(* PLC project Unnamed, Unknown Unnamed 1 *)
(* stored: creationDateTime 2023-06-19T14:42:49, modificationDateTime 2023-08-09T10:28:01 *)

PROGRAM pick_and_place
  VAR
    TP0 : TP;
    CTU0 : CTU;
  END_VAR
  VAR_EXTERNAL
    ITEM_AT_ENTRY : BOOL;
    ITEM_AT_EXIT : BOOL;
    MOVING_X : BOOL;
    MOVING_Z : BOOL;
    ITEM_DETECTED : BOOL;
    START : BOOL;
    RESET : BOOL;
    STOP : BOOL;
    EMERGENCY_STOP : BOOL;
    AUTO : BOOL;
    FACTORY_IO_RUN : BOOL;
    ENTRY_CONVEYOR : BOOL;
    EXIT_CONVEYOR : BOOL;
    MOVE_X : BOOL;
    MOVE_Z : BOOL;
    GRAB : BOOL;
    START_LIGHT : BOOL;
    RESET_LIGHT : BOOL;
    STOP_LIGHT : BOOL;
    start_scada : BOOL;
    reset_scada : BOOL;
    stop_scada : BOOL;
    COUNTER : INT;
  END_VAR
  VAR
    T1_DONE : BOOL;
    TIME_DELAY : TIME := t#3s;
  END_VAR
  VAR_EXTERNAL
    STEP_0 : BOOL;
    STEP_1 : BOOL;
    STEP_2 : BOOL;
    STEP_3 : BOOL;
    STEP_4 : BOOL;
    STEP_5 : BOOL;
    STEP_6 : BOOL;
    STEP_7 : BOOL;
    STEP_LOCATION : INT;
  END_VAR
  VAR  (* added by the conversion: wires and edge detectors of the diagram *)
    R_TRIG1 : R_TRIG;
  END_VAR

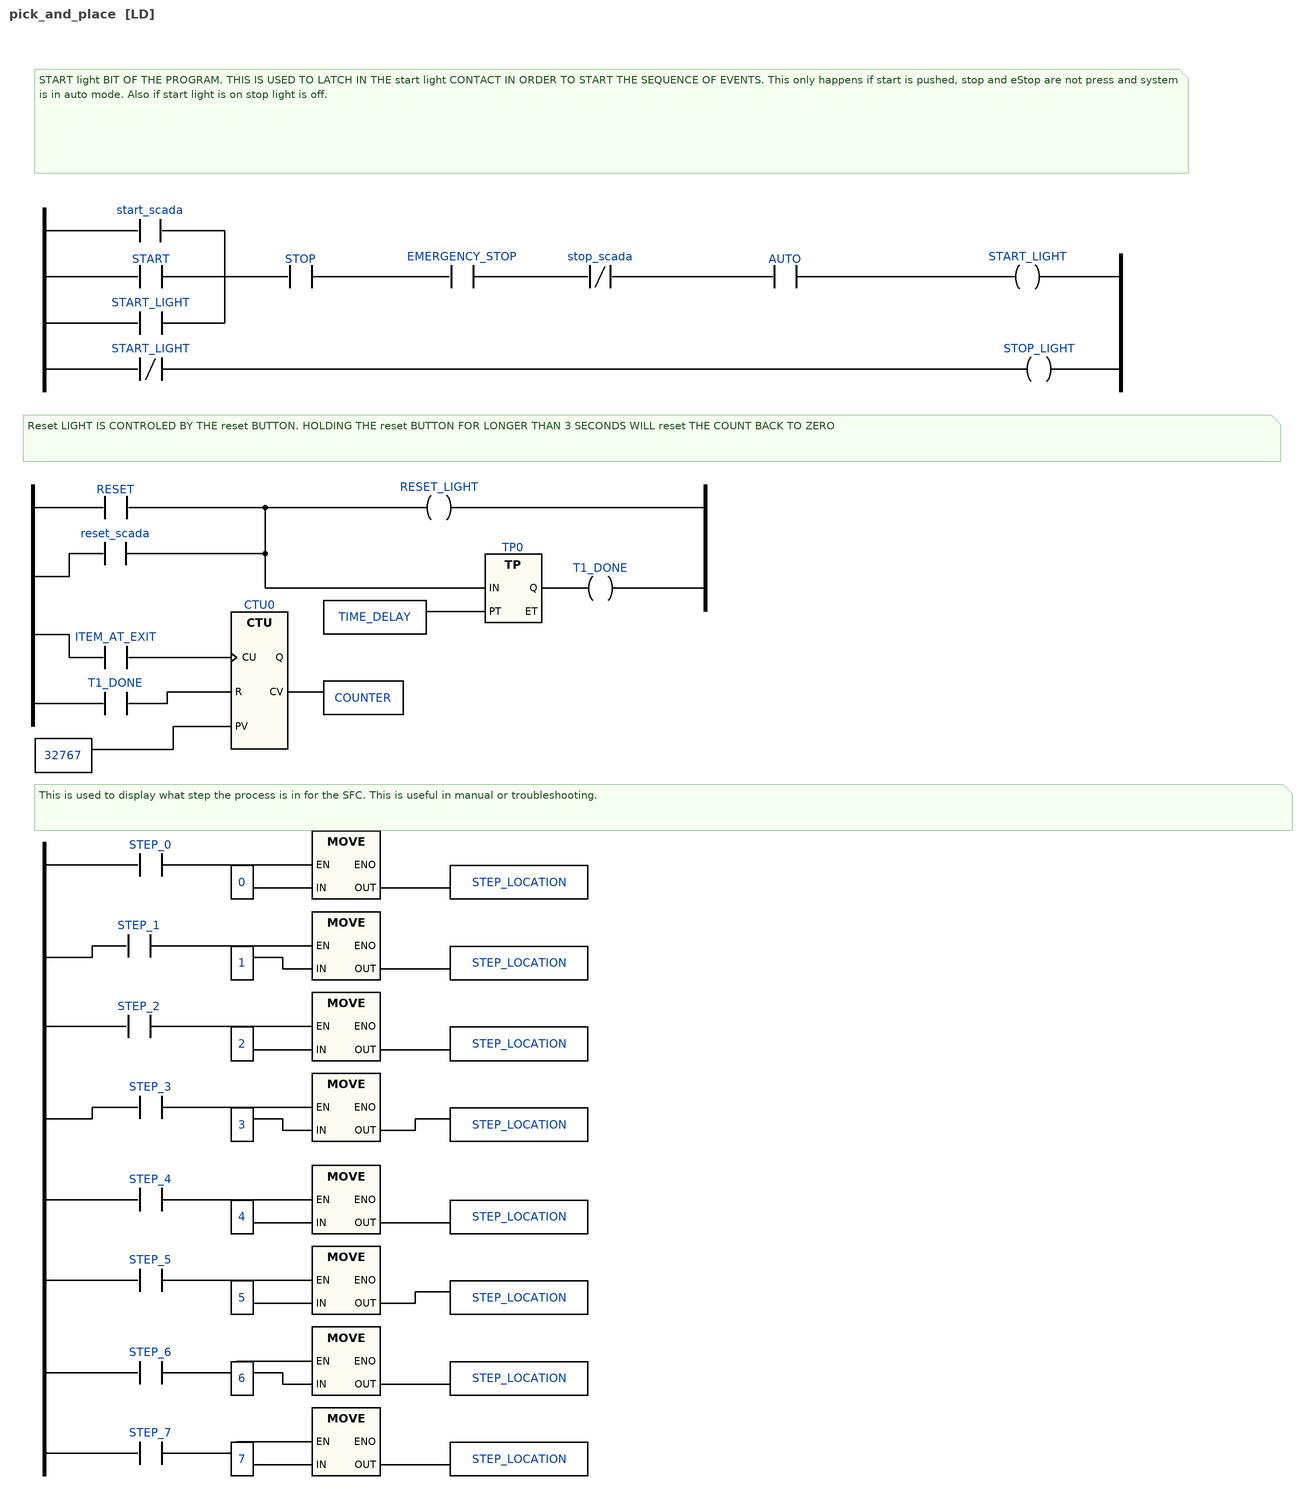
(* LD diagram, written out as Structured Text *)
(* START light BIT OF THE PROGRAM. THIS IS USED TO LATCH IN THE start light CONTACT IN ORDER TO START THE SEQUENCE OF EVENTS. This only happens if start is pushed, stop and eStop are not press and system is in auto mode. Also if start light is on stop light is off. *)
START_LIGHT := (START OR START_LIGHT OR start_scada) AND STOP AND EMERGENCY_STOP AND NOT stop_scada AND AUTO;
STOP_LIGHT := NOT START_LIGHT;
(* Reset LIGHT IS CONTROLED BY THE reset BUTTON. HOLDING THE reset BUTTON FOR LONGER THAN 3 SECONDS WILL reset THE COUNT BACK TO ZERO *)
RESET_LIGHT := RESET OR reset_scada;
TP0(IN := RESET OR reset_scada, PT := TIME_DELAY);
T1_DONE := TP0.Q;
R_TRIG1(CLK := ITEM_AT_EXIT);
CTU0(CU := R_TRIG1.Q, R := T1_DONE, PV := 32767);
COUNTER := CTU0.CV;
(* This is used to display what step the process is in for the SFC. This is useful in manual or troubleshooting. *)
IF STEP_0 THEN STEP_LOCATION := 0; END_IF;
IF STEP_1 THEN STEP_LOCATION := 1; END_IF;
IF STEP_2 THEN STEP_LOCATION := 2; END_IF;
IF STEP_3 THEN STEP_LOCATION := 3; END_IF;
IF STEP_4 THEN STEP_LOCATION := 4; END_IF;
IF STEP_5 THEN STEP_LOCATION := 5; END_IF;
IF STEP_6 THEN STEP_LOCATION := 6; END_IF;
IF STEP_7 THEN STEP_LOCATION := 7; END_IF;
END_PROGRAM

PROGRAM pick_and_place_sfc
  VAR_EXTERNAL
    ITEM_AT_ENTRY : BOOL;
    ITEM_AT_EXIT : BOOL;
    MOVING_X : BOOL;
    MOVING_Z : BOOL;
    ITEM_DETECTED : BOOL;
    START : BOOL;
    RESET : BOOL;
    STOP : BOOL;
    EMERGENCY_STOP : BOOL;
    AUTO : BOOL;
    FACTORY_IO_RUN : BOOL;
    ENTRY_CONVEYOR : BOOL;
    EXIT_CONVEYOR : BOOL;
    MOVE_X : BOOL;
    MOVE_Z : BOOL;
    GRAB : BOOL;
    START_LIGHT : BOOL;
    RESET_LIGHT : BOOL;
    STOP_LIGHT : BOOL;
    STEP_0 : BOOL;
    STEP_1 : BOOL;
    STEP_2 : BOOL;
    STEP_3 : BOOL;
    STEP_4 : BOOL;
    STEP_5 : BOOL;
    STEP_6 : BOOL;
    STEP_7 : BOOL;
    COUNTER : INT;
  END_VAR
  VAR
    R_TRIG0 : R_TRIG;
    F_TRIG0 : F_TRIG;
    F_TRIG1 : F_TRIG;
    F_TRIG2 : F_TRIG;
    F_TRIG3 : F_TRIG;
    F_TRIG4 : F_TRIG;
    F_TRIG5 : F_TRIG;
  END_VAR
  VAR  (* added by the conversion: wires and edge detectors of the diagram *)
    _SEL57_OUT : BOOL;
    _SEL61_OUT : BOOL;
    _SEL64_OUT : BOOL;
    _SEL67_OUT : BOOL;
    _SEL70_OUT : BOOL;
    _SEL73_OUT : BOOL;
    _SEL76_OUT : BOOL;
    _SEL79_OUT : BOOL;
  END_VAR

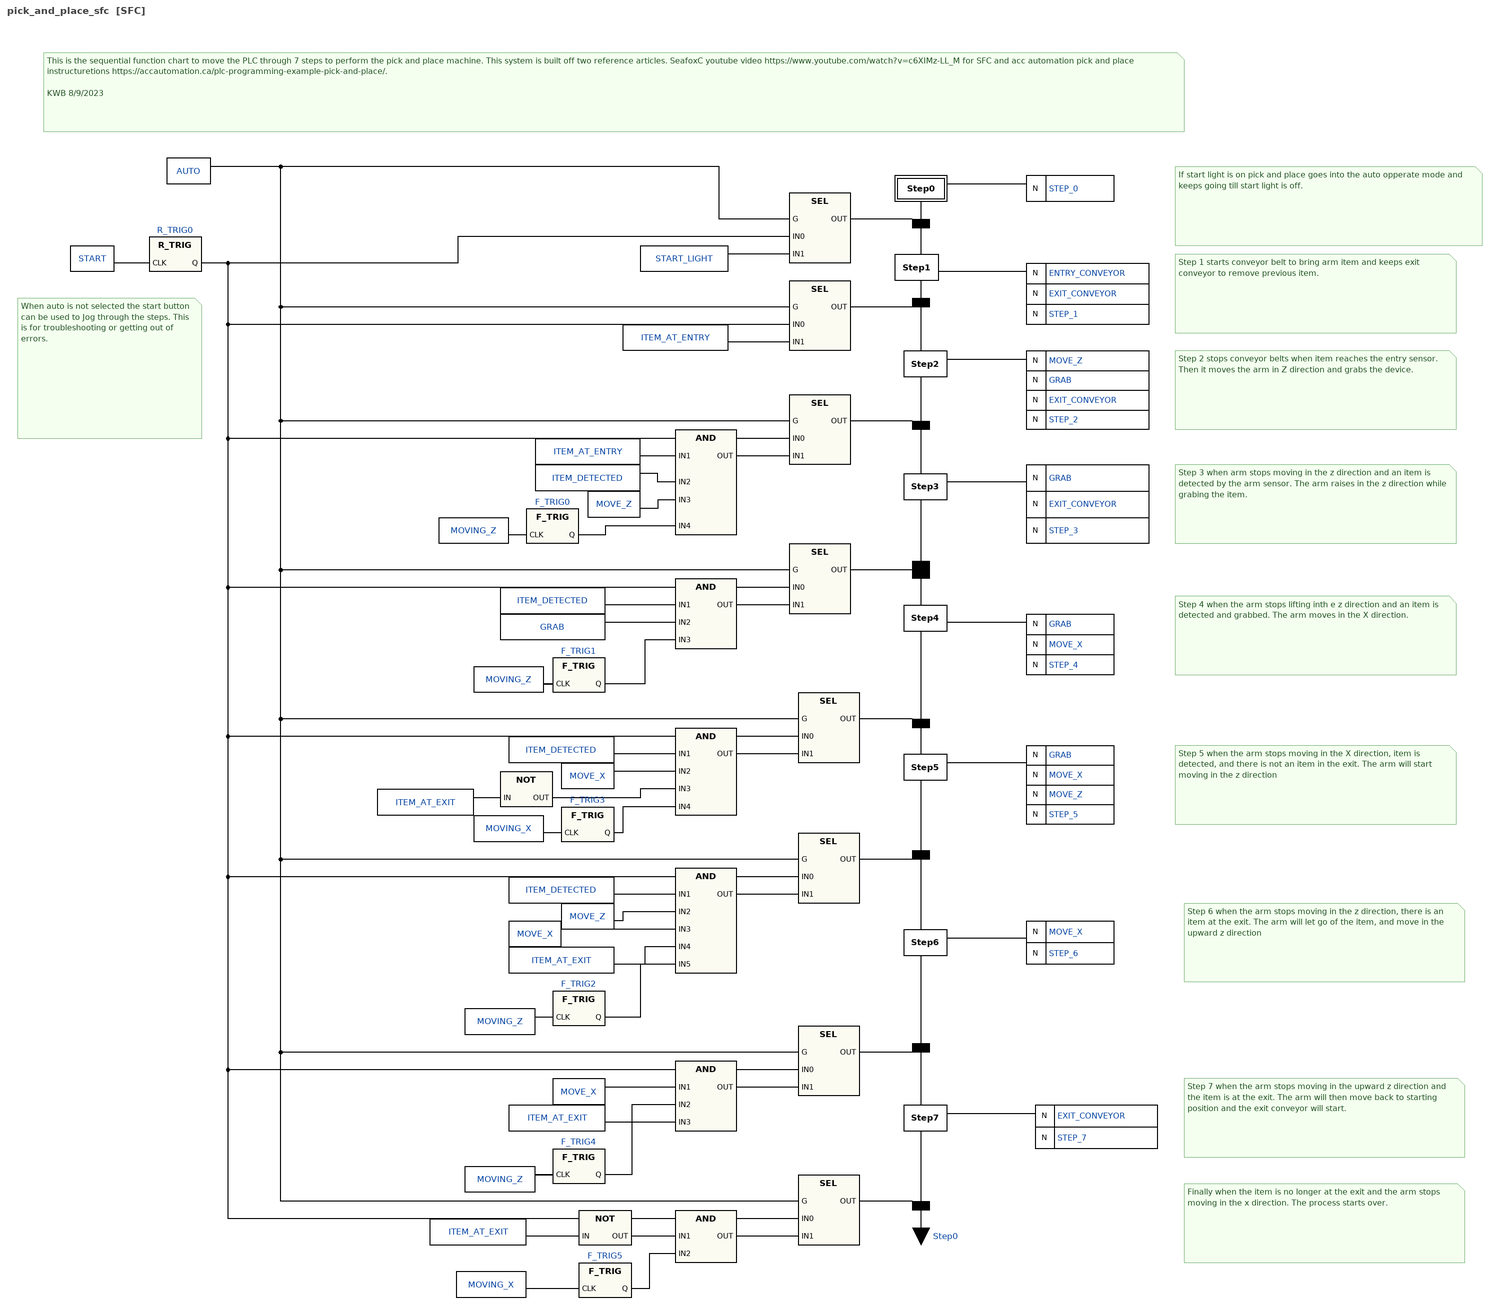
(* When auto is not selected the start button can be used to Jog through the steps. This is for troubleshooting or getting out of errors. *)
(* This is the sequential function chart to move the PLC through 7 steps to perform the pick and place machine. This system is built off two reference articles. SeafoxC youtube video https://www.youtube.com/watch?v=c6XIMz-LL_M for SFC and acc automation pick and place instructuretions https://accautomation.ca/plc-programming-example-pick-and-place/. 

KWB 8/9/2023 *)
(* If start light is on pick and place goes into the auto opperate mode and keeps going till start light is off. *)
(* Step 1 starts conveyor belt to bring arm item and keeps exit conveyor to remove previous item. *)
(* Step 2 stops conveyor belts when item reaches the entry sensor. Then it moves the arm in Z direction and grabs the device. *)
(* Step 3 when arm stops moving in the z direction and an item is detected by the arm sensor. The arm raises in the z direction while grabing the item. *)
(* Step 4 when the arm stops lifting inth e z direction and an item is detected and grabbed. The arm moves in the X direction. *)
(* Step 5 when the arm stops moving in the X direction, item is detected, and there is not an item in the exit. The arm will start moving in the z direction *)
(* Step 6 when the arm stops moving in the z direction, there is an item at the exit. The arm will let go of the item, and move in the upward z direction *)
(* Step 7 when the arm stops moving in the upward z direction and the item is at the exit. The arm will then move back to starting position and the exit conveyor will start. *)
(* Finally when the item is no longer at the exit and the arm stops moving in the x direction. The process starts over. *)
INITIAL_STEP Step0:
  STEP_0(N);
  COMPUTE_FUNCTION_BLOCKS(S);
END_STEP
TRANSITION FROM Step0 TO Step1
  := _SEL57_OUT;
END_TRANSITION
STEP Step1:
  ENTRY_CONVEYOR(N);
  EXIT_CONVEYOR(N);
  STEP_1(N);
END_STEP
TRANSITION FROM Step1 TO Step2
  := _SEL61_OUT;
END_TRANSITION
STEP Step2:
  MOVE_Z(N);
  GRAB(N);
  EXIT_CONVEYOR(N);
  STEP_2(N);
END_STEP
TRANSITION FROM Step2 TO Step3
  := _SEL64_OUT;
END_TRANSITION
STEP Step3:
  GRAB(N);
  EXIT_CONVEYOR(N);
  STEP_3(N);
END_STEP
TRANSITION FROM Step3 TO Step4
  := _SEL67_OUT;
END_TRANSITION
STEP Step4:
  GRAB(N);
  MOVE_X(N);
  STEP_4(N);
END_STEP
TRANSITION FROM Step4 TO Step5
  := _SEL70_OUT;
END_TRANSITION
STEP Step5:
  GRAB(N);
  MOVE_X(N);
  MOVE_Z(N);
  STEP_5(N);
END_STEP
TRANSITION FROM Step5 TO Step6
  := _SEL73_OUT;
END_TRANSITION
STEP Step6:
  MOVE_X(N);
  STEP_6(N);
END_STEP
TRANSITION FROM Step6 TO Step7
  := _SEL76_OUT;
END_TRANSITION
STEP Step7:
  EXIT_CONVEYOR(N);
  STEP_7(N);
END_STEP
TRANSITION FROM Step7 TO Step0
  := _SEL79_OUT;
END_TRANSITION
ACTION COMPUTE_FUNCTION_BLOCKS:  (* blocks drawn on the SFC sheet *)
  R_TRIG0(CLK := START);
  _SEL57_OUT := SEL(AUTO, R_TRIG0.Q, START_LIGHT);
  _SEL61_OUT := SEL(AUTO, R_TRIG0.Q, ITEM_AT_ENTRY);
  F_TRIG0(CLK := MOVING_Z);
  _SEL64_OUT := SEL(AUTO, R_TRIG0.Q, ITEM_AT_ENTRY AND ITEM_DETECTED AND MOVE_Z AND F_TRIG0.Q);
  F_TRIG1(CLK := MOVING_Z);
  _SEL67_OUT := SEL(AUTO, R_TRIG0.Q, ITEM_DETECTED AND GRAB AND F_TRIG1.Q);
  F_TRIG3(CLK := MOVING_X);
  _SEL70_OUT := SEL(AUTO, R_TRIG0.Q, ITEM_DETECTED AND MOVE_X AND NOT ITEM_AT_EXIT AND F_TRIG3.Q);
  F_TRIG2(CLK := MOVING_Z);
  _SEL73_OUT := SEL(AUTO, R_TRIG0.Q, ITEM_DETECTED AND MOVE_Z AND MOVE_X AND ITEM_AT_EXIT AND F_TRIG2.Q);
  F_TRIG4(CLK := MOVING_Z);
  _SEL76_OUT := SEL(AUTO, R_TRIG0.Q, MOVE_X AND ITEM_AT_EXIT AND F_TRIG4.Q);
  F_TRIG5(CLK := MOVING_X);
  _SEL79_OUT := SEL(AUTO, R_TRIG0.Q, NOT ITEM_AT_EXIT AND F_TRIG5.Q);
END_ACTION
END_PROGRAM

CONFIGURATION Config0
  RESOURCE Res0 ON PLC
    VAR_GLOBAL
      ITEM_AT_ENTRY AT %QX0.0 : BOOL;
      ITEM_AT_EXIT AT %QX0.1 : BOOL;
      MOVING_X AT %QX0.2 : BOOL;
      MOVING_Z AT %QX0.3 : BOOL;
      ITEM_DETECTED AT %QX0.4 : BOOL;
      START AT %QX0.5 : BOOL;
      RESET AT %QX0.6 : BOOL;
      STOP AT %QX0.7 : BOOL;
      EMERGENCY_STOP AT %QX1.0 : BOOL;
      AUTO AT %QX1.1 : BOOL;
      FACTORY_IO_RUN AT %QX1.2 : BOOL;
      ENTRY_CONVEYOR AT %QX1.3 : BOOL;
      EXIT_CONVEYOR AT %QX1.4 : BOOL;
      MOVE_X AT %QX1.5 : BOOL;
      MOVE_Z AT %QX1.6 : BOOL;
      GRAB AT %QX1.7 : BOOL;
      START_LIGHT AT %QX2.0 : BOOL;
      RESET_LIGHT AT %QX2.1 : BOOL;
      STOP_LIGHT AT %QX2.2 : BOOL;
      start_scada AT %QX2.3 : BOOL;
      reset_scada AT %QX2.4 : BOOL;
      stop_scada AT %QX2.5 : BOOL;
      COUNTER AT %QW0 : INT;
      STEP_LOCATION AT %QW1 : INT;
      STEP_0 : BOOL;
      STEP_1 : BOOL;
      STEP_2 : BOOL;
      STEP_3 : BOOL;
      STEP_4 : BOOL;
      STEP_5 : BOOL;
      STEP_6 : BOOL;
      STEP_7 : BOOL;
    END_VAR
    TASK task0(INTERVAL := T#20ms, PRIORITY := 0);
    TASK task1(INTERVAL := T#0.1ms, PRIORITY := 0);
    PROGRAM instance0 WITH task0 : pick_and_place;
    PROGRAM instance1 WITH task1 : pick_and_place_sfc;
  END_RESOURCE
END_CONFIGURATION
